(* CODESYS project aliyun.shared-memory.20210305.1.project

Project tree, tasks and I/O mapping:
  Device : Changsha Xiangji-ARM Cortex A9(xilinx zynq7000)-linux, Changsha Xiangji Hiden Technology Co.Ltd, version 3.5.10.40
    application Application
      libraries: Standard, * (System); SysShm, * (System); SysTypes2 Interfaces, * (System); SysFile, 3.5.15.0 (System)
      task MainTask (cyclic, interval 20 ms, priority 10) calls prg_aliyun
      program prg_aliyun [ST]: init, read_from_aliyun, send_to_aliyun
      Struct/
        data type stShmToAliyun
        data type stShmFromAliyun
      global variables GVL
      program prg_printer [ST]
    SoftMotion General Axis Pool
    IoDrvMIC7001 : IoDrvMIC7001, Cyber-MI, version 19.1.1
        unmapped channels: Ai00@C16, Ai01@C28, Ai02@C17, Ai03@C29, Ai04@C30, Ai05@C19, Ai06@C31, Ai07@C20, Ai08@C18, Ai09@D18, Ai10@D20, Ai11@D31, Ai12@D19, Ai13@D30, Ai14@D29, Ai15@D17, Ai16@D28, Ai17@D16, Ai18-Do00@C25, Ai19-Do01@C24, Ai20-Do02@C13, Ai21-Do03@C01, Ai22-Do04@C03, Ai23-Do05@C04, Ai24-Do06@C05, Ai25-Do07@C06, Ai26-Do08@C08, Ai27-Do09@C09, Ai28-Do10@C10, Ai29-Do11@C11, Ai30-Do12@D34, Ai31-Do13@D35, Ai32-Do14@D23, Ai33-Do15@D12, Ai34-Do16@D10, Ai35-Do17@D09, Ai36-Do18@D08, Ai37-Do19@D07, Ai38-Do20@D05, Ai39-Do21@D04,
          Ai40-Do22@D03, Ai41-Do23@D02, Ai42-Do24@C23, Ai43-Do25@C35, Ai44-Do26@D24, Ai45-Do27@D13, Ai46-Ao00@C22, Ai47-Ao01@D14, Ai48_Pi02, Ai49_Out5V, Ai50_VCC, Ai51_VCC_L, Ai52_VCC_R, Ai53_Pwm-i0, Ai54_Pwm-i1, Ai55_Pwm-i2, Ai56_Pwm-i3, Ai57_CPU-T, Ai58_G-x, Ai59_G-y, Ai60_G-z, Ai61-reserved, Ai62-IO-cntr, Ai63-CDS-cntr, Di00-Ai00@C16, Di01-Ai01@C28, Di02-Ai02@C17, Di03-Ai03@C29, Di04-Ai04@C30, Di05-Ai05@C19, Di06-Ai06@C31, Di07-Ai07@C20, Di08-Ai08@C18, Di09-Ai09@D18, Di10-Ai10@D20, Di11-Ai11@D31, Di12-Ai12@D19, Di13-Ai13@D30, Di14-Ai14@D29, Di15-Ai15@D17,
          Di16-Ai16@D28, Di17-Ai17@D16, Di18-Ai18@C25, Di19-Ai19@C24, Di20-Ai20@C13, Di21-Ai21@C01, Di22-Ai22@C03, Di23-Ai23@C04, Di24-Ai24@C05, Di25-Ai25@C06, Di26-Ai26@C08, Di27-Ai27@C09, Di28-Ai28@C10, Di29-Ai29@C11, Di30-Ai30@D34, Di31-Ai31@D35, Di32-Ai32@D23, Di33-Ai33@D12, Di34-Ai34@D10, Di35-Ai35@D09, Di36-Ai36@D08, Di37-Ai37@D07, Di38-Ai38@D05, Di39-Ai39@D04, Di40-Ai40@D03, Di41-Ai41@D02, Di42-Ai42@C23, Di43-Ai43@C35, Di44-Ai44@D24, Di45-Ai45@D13, Di46-Ai46@C22, Di47-Ai47@D14, Di48-Pi00@C15, Di49-Pi01@C14, Di50-Pi02@D22, Di51-Pi03@D21, Di52-reserved, Di53-reserved, Di54-reserved, Di55-reserved,
          Di56-reserved, Di57-reserved, Di58-reserved, Di59-reserved, Di60-reserved, Di61-reserved, Di62-reserved, Di63-reserved, Pi00-Di48@C15, Pi01-Di49@C14, Pi02-Di50@D22, Pi03-Di51@D21, Do00-Ai18@C25, Do01-Ai19@C24, Do02-Ai20@C13, Do03-Ai21@C01, Do04-Ai22@C03, Do05-Ai23@C04, Do06-Ai24@C05, Do07-Ai25@C06, Do08-Ai26@C08, Do09-Ai27@C09, Do10-Ai28@C10, Do11-Ai29@C11, Do12-Ai30@D34, Do13-Ai31@D35, Do14-Ai32@D23, Do15-Ai33@D12, Do16-Ai34@D10, Do17-Ai35@D09, Do18-Ai36@D08, Do19-Ai37@D07, Do20-Ai38@D05, Do21-Ai39@D04, Do22-Ai40@D03, Do23-Ai41@D02, Do24-Ai42@C23, Do25-Ai43@C35, Do26-Ai44@D24, Do27-Ai45@D13,
          Do28-Pwmi00@C33, Do29-Pwmi01@C34, Do30-Pwmi02@D25, Do31-Pwmi03@D26, PWM00@C25, PWM01@C24, PWM02@C13, PWM03@C01, PWM04@C03, PWM05@C04, PWM06@C05, PWM07@C06, PWM08@C08, PWM09@C09, PWM10@C10, PWM11@C11, PWM12@D34, PWM13@D35, PWM14@D23, PWM15@D12, PWM16@D10, PWM17@D09, PWM18@D08, PWM19@D07, PWM20@D05, PWM21@D04, PWM22@D03, PWM23@D02, PWM24@C23, PWM25@C35, PWM26@D24, PWM27@D13, PWM28-Pwmi00@C33, PWM29-Pwmi01@C34, PWM30-Pwmi02@D25, PWM31-Pwmi03@D26, PWM_I_0@C33, PWM_I_1@C34, PWM_I_2@D25, PWM_I_3@D26,
          Ao00-Ai46@C22, Ao01-Ai47@D14, LED_run, LED_err, LED_usr, ctrl_ai_raw, ctrl_adjust, ctrl_adj0, ctrl_adj1, ctrl_adj2, ctrl_adj3, disable_5V
  text list GlobalTextList
  5ce3da45-db07-42e7-a21c-a00fff4ed8f6|C:\Users\pengriguang\Desktop\cyber-tftp\huanweiche.bmp
*)

// Device/Application/Struct/stShmToAliyun
TYPE stShmToAliyun :   // 发送到阿里云物模型的上行数据
STRUCT
    equipment_num :DINT;
    work_state :DINT;
    build_num :DINT;
    pile_num :DINT;
    one_deep :DINT;
    two_deep :DINT;
    three_deep :DINT;
    sum_deep :DINT;
    date_time :DINT;
    lock :DINT;

    time_equipment_num :DINT; // 发送间隔，单位：ms
    time_work_state :DINT;
    time_build_num :DINT;
    time_pile_num :DINT;
    time_one_deep :DINT;
    time_two_deep :DINT;
    time_three_deep :DINT;
    time_sum_deep :DINT;
    time_date_time :DINT;
    time_lock :DINT;
END_STRUCT
END_TYPE

// Device/Application/Struct/stShmFromAliyun
TYPE stShmFromAliyun :  // 从阿里云物模型来的下行数据
STRUCT
	lock:DINT;	 // 锁机命令
END_STRUCT
END_TYPE

// Device/Application/GVL
{attribute 'qualified_only'}
VAR_GLOBAL PERSISTENT RETAIN
	ret_val1: DINT;  
	ret_val2: Dint;
END_VAR

// Device/Application/prg_aliyun
PROGRAM prg_aliyun
VAR
	inited : BOOL := FALSE;
	fluidLow:INT := 0;
	lossWater:INT := 0;
	dirtyWater:INT := 0;
	littleWater:INT := 0;
	pressSuper:INT := 0;
	
	strShmFileDown : STRING := 'SHM_FROM_ALIYUN_7001';
	strShmFileUp : STRING := 'SHM_TO_ALIYUN_7001';
	hShMemDown: RTS_IEC_HANDLE := RTS_INVALID_HANDLE ;
	hShMemUp: RTS_IEC_HANDLE := RTS_INVALID_HANDLE ;
	ResultRead: RTS_IEC_RESULT;
	ResultWrite: RTS_IEC_RESULT;
	
	iRead: __UXINT;
	iWrite: __UXINT;
	shmDataDown:stShmFromAliyun;
	shmDataUp:stShmToAliyun;
	sizeOfStFromAliyun:__UXINT := SIZEOF(stShmFromAliyun);
	sizeOfStToAliyun:__UXINT := SIZEOF(stShmToAliyun);
	
	sim_data : DINT := 0;
	digi_val :DWORD := 0;
	lock_1 :BOOL := FALSE;
	lock_2 :BOOL := FALSE;
	unlock :BOOL := FALSE;
	test_val2 :DINT;
	
	para0:REAL;
	para1:REAL;
	para20:REAL;
	para39:REAL;
END_VAR


IF NOT inited THEN
 	IF NOT init() THEN  // 初始化失败
		RETURN;
	ELSE
		inited := TRUE;
		
		shmDataUp.time_ana_0_19 := 16000;  // 发送周期 16秒
		shmDataUp.time_ana_20_39 := 25000;  // 发送周期 25秒
		shmDataUp.time_ana_40_59 := 25000;  // 发送周期 25秒
		shmDataUp.time_ana_60_79 := 25000;  // 发送周期 25秒
		
		shmDataUp.time_digi_0_29 := 15000;  // 发送周期 15秒
		shmDataUp.time_digi_30_59 := 25000;  // 发送周期 25秒
		shmDataUp.time_digi_60_89 := 35000;  // 发送周期 35秒
		shmDataUp.time_digi_90_119 := 60000;  // 发送周期 1分钟
		
		sim_data := gvl.ret_val1;
		test_val2 := gvl.ret_val2;
	END_IF  
END_IF

IF read_from_aliyun() THEN
   // 读取阿里云发来的数据
	IF shmDataDown.command1 > 0 THEN
		// 处理命令通道1
	END_IF
	
	IF shmDataDown.command2 > 0 THEN
		// 处理命令通道2
	END_IF
	
	IF shmDataDown.digidown_0_29 > 0 THEN
		// 处理下行开关量 0~29
	END_IF
	
	IF shmDataDown.digidown_30_59 > 0 THEN
		// 处理下行开关量 30~59
	END_IF

	// 解析下行参数 0~19
	para0 := shmDataDown.para_0_19[0];  //
	para1 := shmDataDown.para_0_19[1];  //
	// ......
	
	// 解析下行参数 20~39		
	para20 := shmDataDown.para_20_39[0];
	// ......
	para39 := shmDataDown.para_20_39[19];

END_IF

// 准备上传到阿里云的数据
sim_data := sim_data + 1;

(*  ana_0_19
发动机转速
发动机水温
发动机机油压力
发动机燃油箱体积
变速箱涡轮转速
变速箱温度
变速箱压力
吊载重量
前伸距
 臂架角度
臂架长度
刹车油温度
液压油温度
俯仰动作手柄输入
伸缩动作手柄输入
吊具旋转动作输入
吊具侧移动作输入
整机故障代码
*)

shmDataUp.ana_0_19[0] := ANY_TO_REAL(sim_data + 123);
shmDataUp.ana_0_19[3] := ANY_TO_REAL(sim_data + 321);

shmDataUp.ana_20_39[0] := ANY_TO_REAL(sim_data + 1);
shmDataUp.ana_20_39[5] := ANY_TO_REAL(sim_data + 5);
shmDataUp.ana_20_39[12] := ANY_TO_REAL(sim_data + 12);


// ......
shmDataUp.digi_0_29 := 654321;

digi_val.0 := TRUE;
digi_val.2 := FALSE;
digi_val.8 := TRUE;
digi_val.29 := TRUE;  // 最后一个， 30和31不可用
shmDataUp.digi_30_59 := ANY_TO_DINT(digi_val);

shmDataUp.digi_60_89 := 54321;
shmDataUp.digi_90_119 := 4321;


IF sim_data MOD 10000 = 0 THEN
	shmDataUp.error1 :=  shmDataUp.error1 +1;
END_IF

(*
IF sim_data MOD 1000 = 0 THEN
	shmDataUp.error2 := 2002;
END_IF
*)
(*
IF sim_data MOD 1200 = 0 THEN
	shmDataUp.event1 := 3001;
END_IF
*)
(*
IF sim_data MOD 1600 = 0 THEN
	shmDataUp.event2 := 3002;
END_IF
*)
IF send_to_aliyun() THEN
	// write ok
END_IF

METHOD init : bool
VAR_INPUT
END_VAR
init := FALSE;

IF hShMemDown = RTS_INVALID_HANDLE  THEN
	hShMemDown := SysSharedMemoryCreate(strShmFileDown, 0, ADR(sizeOfStFromAliyun), ADR(ResultRead));	
END_IF

IF hShMemUp = RTS_INVALID_HANDLE  THEN
	hShMemUp := SysSharedMemoryCreate(strShmFileUp, 0, ADR(sizeOfStToAliyun), ADR(ResultRead));	
END_IF

IF hShMemDown = RTS_INVALID_HANDLE  OR hShMemUp = RTS_INVALID_HANDLE  THEN
	RETURN;
END_IF

init := TRUE;
RETURN;
END_METHOD

METHOD read_from_aliyun : bool
VAR_INPUT
END_VAR
read_from_aliyun := FALSE;

iRead := SysSharedMemoryRead(hShMemDown, 0, ADR(shmDataDown), sizeOfStFromAliyun, ADR(ResultRead));
IF iRead = sizeOfStFromAliyun THEN
    read_from_aliyun := TRUE;
END_IF

RETURN;
END_METHOD

METHOD send_to_aliyun : bool
VAR_INPUT
END_VAR
send_to_aliyun := FALSE;

iWrite := SysSharedMemoryWrite(hShMemUp, 0, ADR(shmDataUp), sizeOfStToAliyun, ADR(ResultWrite));
IF iWrite = sizeOfStToAliyun THEN
	send_to_aliyun := TRUE;
END_IF

RETURN;
END_METHOD

END_PROGRAM

// Device/Application/prg_printer
PROGRAM prg_printer
VAR
	filename:STRING := '/dev/usb/lp0';
	hFile: RTS_IEC_HANDLE := 0;
	udiOpenError:RTS_IEC_RESULT;
	udiWriteError:RTS_IEC_RESULT;
	
	stat:DINT := 0;
	
	str_print:STRING(255);
	cmd_print:BOOL := FALSE;
END_VAR


CASE stat OF
0:
	hFile := sysfileopen(szFile := filename, am := sysfile.AM_WRITE, pResult:= ADR(udiOpenError));
	IF hFile = RTS_INVALID_HANDLE THEN
		RETURN;
	ELSE
		stat := 10;
    END_IF

10:  //waite print command
    IF cmd_print THEN
		sysfilewrite(hFile := hFile, pbyBuffer := ADR(str_print), ulSize := len(str_print), pResult := ADR(udiWriteError));
		cmd_print := FALSE;
	END_IF
END_CASE

END_PROGRAM
